FUNCTION_BLOCK Humano IMPLEMENTS I_Humano
VAR_INPUT
END_VAR
VAR_OUTPUT
END_VAR
VAR
END_VAR

{warning 'Agregar implementación de método'}
METHOD Correr
END_METHOD

{warning 'Agregar implementación de propiedad'}
PROPERTY Nombre : STRING
GET
END_GET
SET
END_SET
END_PROPERTY

END_FUNCTION_BLOCK

(* stored: Version 1.1.0.1, ProductVersion 3.1.4024.12
   POU Humano: Id {d4a32384-1ff2-4dfd-8276-2238a328a67c}, SpecialFunc None
   Method Correr: Id {ab751311-0c3f-42a9-aced-90d53b2c17b9}
   Property Nombre: Id {e40449f4-a3e0-409c-92f6-4841bff99f06}
   Get Get: Id {0beb7bab-28f8-4ee2-a443-6e46b3829b63}
   Set Set: Id {a701ccd5-5fdb-423c-9b59-1206c62c592b} *)
